// TIA Portal V16 export
// export: Created 2023-01-04T15:44:09.7043887Z, ExportSetting WithDefaults, DisplayName Totally Integrated Automation Portal, DisplayVersion V16, DisplayName TIA Portal Version Control Interface, DisplayVersion V16, DisplayName TIA Portal Openness, DisplayVersion V16, DisplayName STEP 7 Professional, DisplayVersion V16, DisplayName STEP 7 Safety, DisplayVersion V16, DisplayName WinCC Advanced, DisplayVersion V16
DATA_BLOCK "Global_DB"   // DB1
{ S7_Optimized_Access := 'TRUE' }
VERSION : 0.1
// stored: AutoNumber true, DBAccessibleFromOPCUA true, IsOnlyStoredInLoadMemory false, IsRetainMemResEnabled false, IsWriteProtectedInAS false, MemoryReserve 100
   VAR
      Input : Struct
         FIC_B102 : Int;   // Tank2 Level Measurement
         LIC_B101 : Int;
         PS1_RFID_Station : Bool;
         PS2_Filling_Station : Bool;
         PS3_Quality_Station : Bool;
         PS4_End_of_Conveyor : Bool;
         T01_Low_Level : Bool;
         T01_High_Level : Bool;
      END_STRUCT;
      Output : Struct
         T01_Outlet : Bool;
         T02_Outlet : Bool;
         Outlet_Pump_Motor : Bool;
         Conveyor_Motor : Bool;
         T01_Inlet : Bool;
         T02_Inlet : Bool;
      END_STRUCT;
      Other_Parameters : Struct
         Liquid_A_Filled : Bool;
         Add_Done : Bool;
         Liquid_B_Filled : Bool;
         Flow_ml_per_sec : Real;
         LiquidA_in_Bottle_ml : Real;
         LiquidB_in_Bottle_ml : Real;
         T02_Level_in_L : Real;
         T02_High_Level_Limit { ExternalVisible := 'False'} : Real;
         T02_Low_Level_Limit : Real;
         Liquid_A_pct : Int := 50;   // data from RFID tags
         Liquid_B_pct : Int := 50;   // datafrom RFID tags
         Alarm_Reset : Bool;
         operation_cycle_time : Time;
         index : Int := 1;
      END_STRUCT;
      Error : Struct
         Alarm : Word;
      END_STRUCT;
      Master_Command : Struct
         operation_begin : Bool;
         operation_finished : Bool;
      END_STRUCT;
      Production_Data : Struct   // Unit ml
         Total_Liquid_in_Bottle : Array[1..5] of Real;
         LiquidA_in_Bottle : Array[1..5] of Real;
         operation_cycles : Array[1..5] of Time;
         LiquidB_in_Bottle : Array[1..5] of Real;
         current_cycle : Int := 1;
         Bottle_Count : Int := 1;   // Total Bottle filled
      END_STRUCT;
   END_VAR
BEGIN
END_DATA_BLOCK
